// TIA Portal V17 export
// export: Created 2024-09-02T12:49:54.0325242Z, ExportSetting WithDefaults, DisplayName Totally Integrated Automation Portal, DisplayVersion V17, DisplayName TIA Portal Openness, DisplayVersion V17, DisplayName TIA Portal Version Control Interface, DisplayVersion V17, DisplayName STEP 7 Professional, DisplayVersion V17, DisplayName STEP 7 Safety, DisplayVersion V17, DisplayName WinCC Professional, DisplayVersion V17
FUNCTION_BLOCK "AnwFB_Safety"   // FB7001, F_LAD
TITLE = Safety program / Safety-Programm
{ S7_Optimized_Access := 'TRUE' }
AUTHOR : OlegFuehrus
FAMILY : SAFETY
NAME : SAFETY
VERSION : 0.1
// stored: AutoNumber false, IsIECCheckEnabled false, UDAEnableTagReadback false
   VAR
      statTrue : Bool := true;   // TRUE
      statFalse : Bool := false;   // FALSE
      HM_1_ack : Bool;   // Hilfvar Quittieren / Hilfvar Acknowledge
      HM_SK_ack_1 : Bool;   // Hilfvar Quittieren Schutzkreise / Hilfvar Acknowledge Protective circuits
      HM_FGroup_ack : Bool;   // Hilfvar Quittieren F-Baugruppen / Hilfvar Acknowledge F assemblies
      HM_LC_ack_1 : Bool;   // Hilfvar Quittieren Lichtgitter / Hilfvar Acknowledge Light grid
      Error_FDback_all { ExternalWritable := 'False'} : Bool;   // Fehler FDBack / Error FDBack
      ACK_Global { S7_SetPoint := 'True'} : ACK_GL;   // ACK Global
      EStop_1 { S7_SetPoint := 'True'} : ESTOP1;   // Not-Halt / emergency stop
      EStop_2 { S7_SetPoint := 'True'} : ESTOP1;   // Not-Halt / emergency stop
      EStop_3 { S7_SetPoint := 'True'} : ESTOP1;   // Not-Halt / emergency stop
      EStop_4 { S7_SetPoint := 'True'} : ESTOP1;   // Not-Halt / emergency stop
      EStop_5 { S7_SetPoint := 'True'} : ESTOP1;   // Not-Halt / emergency stop
      EStop_6 { S7_SetPoint := 'True'} : ESTOP1;   // Not-Halt / emergency stop
      EStop_7 { S7_SetPoint := 'True'} : ESTOP1;   // Not-Halt / emergency stop
      EStop_8 { S7_SetPoint := 'True'} : ESTOP1;   // Not-Halt / emergency stop
      LC_1 { S7_SetPoint := 'True'} : ESTOP1;   // Lichtgitter / light curtain
      LC_2 { S7_SetPoint := 'True'} : ESTOP1;   // Lichtgitter / light curtain
      LC_3 { S7_SetPoint := 'True'} : ESTOP1;   // Lichtgitter / light curtain
      LC_4 { S7_SetPoint := 'True'} : ESTOP1;   // Lichtgitter / light curtain
      LC_5 { S7_SetPoint := 'True'} : ESTOP1;   // Lichtgitter / light curtain
      LC_MUT_1 { S7_SetPoint := 'True'} : MUT_P;   // Lichtgitter mit Muting / Light curtain with muting
      LC_MUT_2 { S7_SetPoint := 'True'} : MUT_P;   // Lichtgitter mit Muting / Light curtain with muting
      LC_MUT_3 { S7_SetPoint := 'True'} : MUT_P;   // Lichtgitter mit Muting / Light curtain with muting
      LC_MUT_4 { S7_SetPoint := 'True'} : MUT_P;   // Lichtgitter mit Muting / Light curtain with muting
      LC_MUT_5 { S7_SetPoint := 'True'} : MUT_P;   // Lichtgitter mit Muting / Light curtain with muting
      SD_1 { S7_SetPoint := 'True'} : ESTOP1;   // Schutzgitter / Safety guard
      SD_2 { S7_SetPoint := 'True'} : ESTOP1;   // Schutzgitter / Safety guard
      SD_3 { S7_SetPoint := 'True'} : ESTOP1;   // Schutzgitter / Safety guard
      SD_4 { S7_SetPoint := 'True'} : ESTOP1;   // Schutzgitter / Safety guard
      SD_5 { S7_SetPoint := 'True'} : ESTOP1;   // Schutzgitter / Safety guard
      BR_1 { S7_SetPoint := 'True'} : EV1oo2DI;   // Überbrückung / Bridging
      BR_2 { S7_SetPoint := 'True'} : EV1oo2DI;   // Überbrückung / Bridging
      BR_3 { S7_SetPoint := 'True'} : EV1oo2DI;   // Überbrückung / Bridging
      BR_4 { S7_SetPoint := 'True'} : EV1oo2DI;   // Überbrückung / Bridging
      BR_5 { S7_SetPoint := 'True'} : EV1oo2DI;   // Überbrückung / Bridging
      EnblCircuit_01 { S7_SetPoint := 'True'} : FDBACK;   // Freigabekreis / Relase circuit
      EnblCircuit_02 { S7_SetPoint := 'True'} : FDBACK;   // Freigabekreis / Relase circuit
      EnblCircuit_03 { S7_SetPoint := 'True'} : FDBACK;   // Freigabekreis / Relase circuit
      EnblCircuit_04 { S7_SetPoint := 'True'} : FDBACK;   // Freigabekreis / Relase circuit
      EnblCircuit_05 { S7_SetPoint := 'True'} : FDBACK;   // Freigabekreis / Relase circuit
      EnblCircuit_06 { S7_SetPoint := 'True'} : FDBACK;   // Freigabekreis / Relase circuit
      EnblCircuit_07 { S7_SetPoint := 'True'} : FDBACK;   // Freigabekreis / Relase circuit
      EnblCircuit_08 { S7_SetPoint := 'True'} : FDBACK;   // Freigabekreis / Relase circuit
      EnblCircuit_09 { S7_SetPoint := 'True'} : FDBACK;   // Freigabekreis / Relase circuit
      EnblCircuit_10 { S7_SetPoint := 'True'} : FDBACK;   // Freigabekreis / Relase circuit
      EnblCircuit_11 { S7_SetPoint := 'True'} : FDBACK;   // Freigabekreis / Relase circuit
      EnblCircuit_12 { S7_SetPoint := 'True'} : FDBACK;   // Freigabekreis / Relase circuit
      EnblCircuit_13 { S7_SetPoint := 'True'} : FDBACK;   // Freigabekreis / Relase circuit
      EnblCircuit_14 { S7_SetPoint := 'True'} : FDBACK;   // Freigabekreis / Relase circuit
      EnblCircuit_15 { S7_SetPoint := 'True'} : FDBACK;   // Freigabekreis / Relase circuit
      SafetyZone_1 { S7_SetPoint := 'True'} : EV1oo2DI;   // Schutzbereich / Scope of protection
      SafetyZone_2 { S7_SetPoint := 'True'} : EV1oo2DI;   // Schutzbereich / Scope of protection
      SafetyZone_3 { S7_SetPoint := 'True'} : EV1oo2DI;   // Schutzbereich / Scope of protection
      SafetyZone_4 { S7_SetPoint := 'True'} : EV1oo2DI;   // Schutzbereich / Scope of protection
      SafetyZone_5 { S7_SetPoint := 'True'} : EV1oo2DI;   // Schutzbereich / Scope of protection
      EnblCircuit_delay_01 { S7_SetPoint := 'True'} : TOF;   // Freigabekreis verzoegert / Release circuit delayed
      EnblCircuit_delay_02 { S7_SetPoint := 'True'} : TOF;   // Freigabekreis verzoegert / Release circuit delayed
      EnblCircuit_delay_03 { S7_SetPoint := 'True'} : TOF;   // Freigabekreis verzoegert / Release circuit delayed
      EnblCircuit_delay_04 { S7_SetPoint := 'True'} : TOF;   // Freigabekreis verzoegert / Release circuit delayed
      EnblCircuit_delay_05 { S7_SetPoint := 'True'} : TOF;   // Freigabekreis verzoegert / Release circuit delayed
      EnblCircuit_delay_06 { S7_SetPoint := 'True'} : TOF;   // Freigabekreis verzoegert / Release circuit delayed
      EnblCircuit_delay_07 { S7_SetPoint := 'True'} : TOF;   // Freigabekreis verzoegert / Release circuit delayed
      EnblCircuit_delay_08 { S7_SetPoint := 'True'} : TOF;   // Freigabekreis verzoegert / Release circuit delayed
      EnblCircuit_delay_09 { S7_SetPoint := 'True'} : TOF;   // Freigabekreis verzoegert / Release circuit delayed
      EnblCircuit_delay_10 { S7_SetPoint := 'True'} : TOF;   // Freigabekreis verzoegert / Release circuit delayed
      EnblCircuit_delay_11 { S7_SetPoint := 'True'} : TOF;   // Freigabekreis verzoegert / Release circuit delayed
      EnblCircuit_delay_12 { S7_SetPoint := 'True'} : TOF;   // Freigabekreis verzoegert / Release circuit delayed
      EnblCircuit_delay_13 { S7_SetPoint := 'True'} : TOF;   // Freigabekreis verzoegert / Release circuit delayed
      EnblCircuit_delay_14 { S7_SetPoint := 'True'} : TOF;   // Freigabekreis verzoegert / Release circuit delayed
      EnblCircuit_delay_15 { S7_SetPoint := 'True'} : TOF;   // Freigabekreis verzoegert / Release circuit delayed
   END_VAR
   VAR_TEMP
      t_VKE0 : Bool;   // VKE0
      t_VKE1 : Bool;   // VKE1
      t_dummy : Bool;   // Dummy
      t_startcond_1 : Bool;   // Startvorrausetzung / starting prerequisite
      t_startcond_2 : Bool;
      t_fp_ack : Bool;   // Flanke Quit / Flank Quit
      t_fp_SQ_ack_2 : Bool;   // Flanke Quit Schutzkreis / Flank Quit protection circuit
      t_fp_SQ_ack_1 : Bool;   // Flanke Quit Schutzkreis / Flank Quit protection circuit
      t_fp_SQ_error_ack_2 : Bool;   // Flanke Quit Schutzkreis ohne Fehler / Flank Quit Protective circuit without fault
      t_fp_SQ_error_ack_1 : Bool;   // Flanke Quit Schutzkreis ohne Fehler / Flank Quit Protective circuit without fault
      t_fp_FGroup_ack_2 : Bool;   // Flanke Quit F-Baugruppen / Flank Quit F assemblies
      t_fp_FGroup_ack_1 : Bool;   // Flanke Quit F-Baugruppen / Flank Quit F assemblies
      t_fp_LC_ack_1 : Bool;   // Flanke Quit Lichtgitter / Flank Quit light grid
      t_EStopModule : Bool;
   END_VAR
   VAR_TEMP   // added for the SCL form of the ladder/FBD networks
      _w1 : Bool;
   END_VAR
BEGIN

REGION Network 1: VKE 0/1
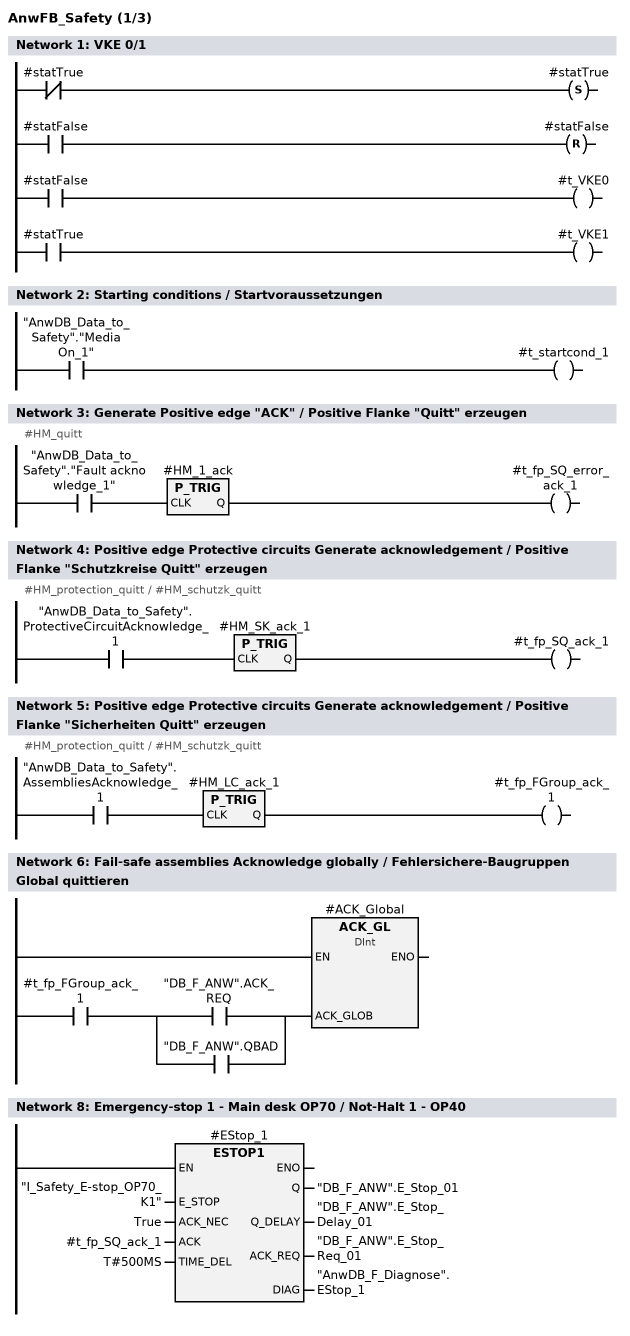
   RUNG wire#powerrail
      I_Contact( #statTrue )
      S_Coil( #statTrue )
   END_RUNG
   RUNG wire#powerrail
      Contact( #statFalse )
      R_Coil( #statFalse )
   END_RUNG
   RUNG wire#powerrail
      Contact( #statFalse )
      Coil( #t_VKE0 )
   END_RUNG
   RUNG wire#powerrail
      Contact( #statTrue )
      Coil( #t_VKE1 )
   END_RUNG
   // the same network as SCL:
   IF NOT #statTrue THEN #statTrue := TRUE; END_IF;
   IF #statFalse THEN #statFalse := FALSE; END_IF;
   #t_VKE0 := #statFalse;
   #t_VKE1 := #statTrue;
END_REGION

REGION Network 2: Starting conditions / Startvoraussetzungen
   RUNG wire#powerrail
      Contact( "AnwDB_Data_to_Safety"."Media On_1" )
      Coil( #t_startcond_1 )
   END_RUNG
   // the same network as SCL:
   #t_startcond_1 := "AnwDB_Data_to_Safety"."Media On_1";
END_REGION

REGION Network 3: Generate Positive edge "ACK" / Positive Flanke "Quitt" erzeugen
   // #HM_quitt
   RUNG wire#powerrail
      Contact( "AnwDB_Data_to_Safety"."Fault acknowledge_1" )
      P_Trig( #HM_1_ack )
      Coil( #t_fp_SQ_error_ack_1 )
   END_RUNG
   // the same network as SCL:
   #_w1 := "AnwDB_Data_to_Safety"."Fault acknowledge_1" AND NOT #HM_1_ack;   // rising edge
   #HM_1_ack := "AnwDB_Data_to_Safety"."Fault acknowledge_1";
   #t_fp_SQ_error_ack_1 := #_w1;
END_REGION

REGION Network 4: Positive edge Protective circuits Generate acknowledgement / Positive Flanke "Schutzkreise Quitt" erzeugen
   // #HM_protection_quitt / #HM_schutzk_quitt
   RUNG wire#powerrail
      Contact( "AnwDB_Data_to_Safety".ProtectiveCircuitAcknowledge_1 )
      P_Trig( #HM_SK_ack_1 )
      Coil( #t_fp_SQ_ack_1 )
   END_RUNG
   // the same network as SCL:
   #_w1 := "AnwDB_Data_to_Safety".ProtectiveCircuitAcknowledge_1 AND NOT #HM_SK_ack_1;   // rising edge
   #HM_SK_ack_1 := "AnwDB_Data_to_Safety".ProtectiveCircuitAcknowledge_1;
   #t_fp_SQ_ack_1 := #_w1;
END_REGION

REGION Network 5: Positive edge Protective circuits Generate acknowledgement / Positive Flanke "Sicherheiten Quitt" erzeugen
   // #HM_protection_quitt / #HM_schutzk_quitt
   RUNG wire#powerrail
      Contact( "AnwDB_Data_to_Safety".AssembliesAcknowledge_1 )
      P_Trig( #HM_LC_ack_1 )
      Coil( #t_fp_FGroup_ack_1 )
   END_RUNG
   // the same network as SCL:
   #_w1 := "AnwDB_Data_to_Safety".AssembliesAcknowledge_1 AND NOT #HM_LC_ack_1;   // rising edge
   #HM_LC_ack_1 := "AnwDB_Data_to_Safety".AssembliesAcknowledge_1;
   #t_fp_FGroup_ack_1 := #_w1;
END_REGION

REGION Network 6: Fail-safe assemblies Acknowledge globally / Fehlersichere-Baugruppen Global quittieren
   RUNG wire#powerrail
      { S7_Templates := "codedbool_type := DInt" } #ACK_Global.ACK_GL(ACK_GLOB := wire#w2)
   END_RUNG
   RUNG wire#powerrail
      Contact( #t_fp_FGroup_ack_1 )
      wire#w1
      Contact( "DB_F_ANW".ACK_REQ )
   END_RUNG wire#w2
   RUNG wire#w1
      Contact( "DB_F_ANW".QBAD )
   END_RUNG wire#w2
   // the same network as SCL:
   #ACK_Global(ACK_GLOB := #t_fp_FGroup_ack_1 AND ("DB_F_ANW".ACK_REQ OR "DB_F_ANW".QBAD));   // ACK_GL
END_REGION

REGION Network 7: ############# ACTUATORS ############## / ######################### AKTOREN ########################
END_REGION

REGION Network 8: Emergency-stop 1 - Main desk OP70 / Not-Halt 1 - OP40
   RUNG wire#powerrail
      #EStop_1.ESTOP1(E_STOP := "I_Safety_E-stop_OP70_K1", ACK_NEC := True, ACK := #t_fp_SQ_ack_1, TIME_DEL := T#500MS, Q => "DB_F_ANW".E_Stop_01, Q_DELAY => "DB_F_ANW".E_Stop_Delay_01, ACK_REQ => "DB_F_ANW".E_Stop_Req_01, DIAG => "AnwDB_F_Diagnose".EStop_1)
   END_RUNG
   // the same network as SCL:
   #EStop_1(E_STOP := "I_Safety_E-stop_OP70_K1",   // ESTOP1
            ACK_NEC := True,
            ACK := #t_fp_SQ_ack_1,
            TIME_DEL := T#500MS,
            Q => "DB_F_ANW".E_Stop_01,
            Q_DELAY => "DB_F_ANW".E_Stop_Delay_01,
            ACK_REQ => "DB_F_ANW".E_Stop_Req_01,
            DIAG => "AnwDB_F_Diagnose".EStop_1);
END_REGION

REGION Network 9: Emergency stop OK. / Not-Halt i.O.
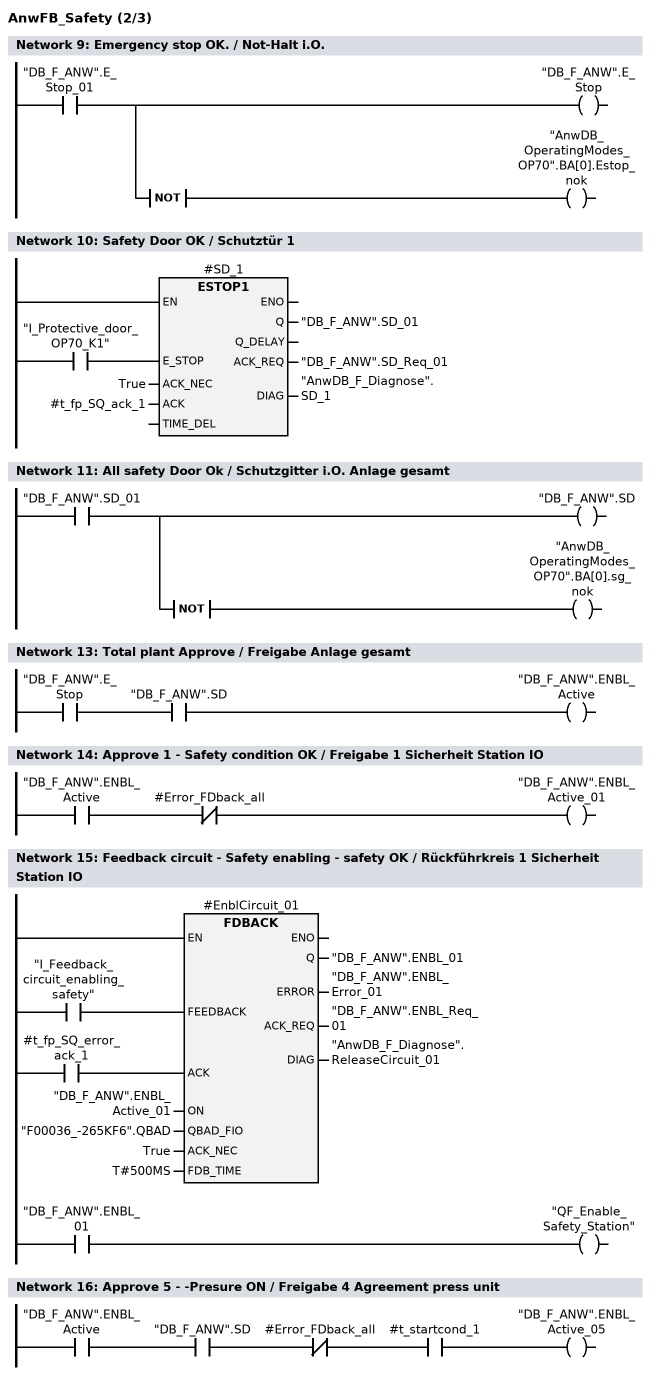
   RUNG wire#powerrail
      Contact( "DB_F_ANW".E_Stop_01 )
      wire#w1
      Coil( "DB_F_ANW".E_Stop )
   END_RUNG
   RUNG wire#w1
      Not()
      Coil( "AnwDB_OperatingModes_OP70".BA[0].Estop_nok )
   END_RUNG
   // the same network as SCL:
   "DB_F_ANW".E_Stop := "DB_F_ANW".E_Stop_01;
   "AnwDB_OperatingModes_OP70".BA[0].Estop_nok := NOT "DB_F_ANW".E_Stop_01;
END_REGION

REGION Network 10: Safety Door OK / Schutztür 1
   RUNG wire#powerrail
      #SD_1.ESTOP1(E_STOP := wire#w1, ACK_NEC := True, ACK := #t_fp_SQ_ack_1, TIME_DEL :=, Q => "DB_F_ANW".SD_01, Q_DELAY =>, ACK_REQ => "DB_F_ANW".SD_Req_01, DIAG => "AnwDB_F_Diagnose".SD_1)
   END_RUNG
   RUNG wire#powerrail
      Contact( "I_Protective_door_OP70_K1" )
   END_RUNG wire#w1
   // the same network as SCL:
   #SD_1(E_STOP := "I_Protective_door_OP70_K1",   // ESTOP1
         ACK_NEC := True,
         ACK := #t_fp_SQ_ack_1,
         Q => "DB_F_ANW".SD_01,
         ACK_REQ => "DB_F_ANW".SD_Req_01,
         DIAG => "AnwDB_F_Diagnose".SD_1);
END_REGION

REGION Network 11: All safety Door Ok / Schutzgitter i.O. Anlage gesamt
   RUNG wire#powerrail
      Contact( "DB_F_ANW".SD_01 )
      wire#w1
      Coil( "DB_F_ANW".SD )
   END_RUNG
   RUNG wire#w1
      Not()
      Coil( "AnwDB_OperatingModes_OP70".BA[0].sg_nok )
   END_RUNG
   // the same network as SCL:
   "DB_F_ANW".SD := "DB_F_ANW".SD_01;
   "AnwDB_OperatingModes_OP70".BA[0].sg_nok := NOT "DB_F_ANW".SD_01;
END_REGION

REGION Network 12: ############# PERMISIIONS ############## / ######################### FREIGABEN ########################
END_REGION

REGION Network 13: Total plant Approve / Freigabe Anlage gesamt
   RUNG wire#powerrail
      Contact( "DB_F_ANW".E_Stop )
      Contact( "DB_F_ANW".SD )
      Coil( "DB_F_ANW".ENBL_Active )
   END_RUNG
   // the same network as SCL:
   "DB_F_ANW".ENBL_Active := "DB_F_ANW".E_Stop AND "DB_F_ANW".SD;
END_REGION

REGION Network 14: Approve 1 - Safety condition OK / Freigabe 1 Sicherheit Station IO
   RUNG wire#powerrail
      Contact( "DB_F_ANW".ENBL_Active )
      I_Contact( #Error_FDback_all )
      Coil( "DB_F_ANW".ENBL_Active_01 )
   END_RUNG
   // the same network as SCL:
   "DB_F_ANW".ENBL_Active_01 := "DB_F_ANW".ENBL_Active AND NOT #Error_FDback_all;
END_REGION

REGION Network 15: Feedback circuit - Safety enabling - safety OK / Rückführkreis 1 Sicherheit Station IO
   RUNG wire#powerrail
      #EnblCircuit_01.FDBACK(FEEDBACK := wire#w1, ACK := wire#w2, ON := "DB_F_ANW".ENBL_Active_01, QBAD_FIO := "F00036_-265KF6".QBAD, ACK_NEC := True, FDB_TIME := T#500MS, Q => "DB_F_ANW".ENBL_01, ERROR => "DB_F_ANW".ENBL_Error_01, ACK_REQ => "DB_F_ANW".ENBL_Req_01, DIAG => "AnwDB_F_Diagnose".ReleaseCircuit_01)
   END_RUNG
   RUNG wire#powerrail
      Contact( "I_Feedback_circuit_enabling_safety" )
   END_RUNG wire#w1
   RUNG wire#powerrail
      Contact( #t_fp_SQ_error_ack_1 )
   END_RUNG wire#w2
   RUNG wire#powerrail
      Contact( "DB_F_ANW".ENBL_01 )
      Coil( "QF_Enable_Safety_Station" )
   END_RUNG
   // the same network as SCL:
   #EnblCircuit_01(FEEDBACK := "I_Feedback_circuit_enabling_safety",   // FDBACK
                   ACK := #t_fp_SQ_error_ack_1,
                   ON := "DB_F_ANW".ENBL_Active_01,
                   QBAD_FIO := "F00036_-265KF6".QBAD,
                   ACK_NEC := True,
                   FDB_TIME := T#500MS,
                   Q => "DB_F_ANW".ENBL_01,
                   ERROR => "DB_F_ANW".ENBL_Error_01,
                   ACK_REQ => "DB_F_ANW".ENBL_Req_01,
                   DIAG => "AnwDB_F_Diagnose".ReleaseCircuit_01);
   "QF_Enable_Safety_Station" := "DB_F_ANW".ENBL_01;
END_REGION

REGION Network 16: Approve 5 - -Presure ON / Freigabe 4 Agreement press unit
   RUNG wire#powerrail
      Contact( "DB_F_ANW".ENBL_Active )
      Contact( "DB_F_ANW".SD )
      I_Contact( #Error_FDback_all )
      Contact( #t_startcond_1 )
      Coil( "DB_F_ANW".ENBL_Active_05 )
   END_RUNG
   // the same network as SCL:
   "DB_F_ANW".ENBL_Active_05 := "DB_F_ANW".ENBL_Active AND "DB_F_ANW".SD AND NOT #Error_FDback_all AND #t_startcond_1;
END_REGION

REGION Network 17: Feedback circuit - Presure ON / Rückführkreis 2 Not Halt IO
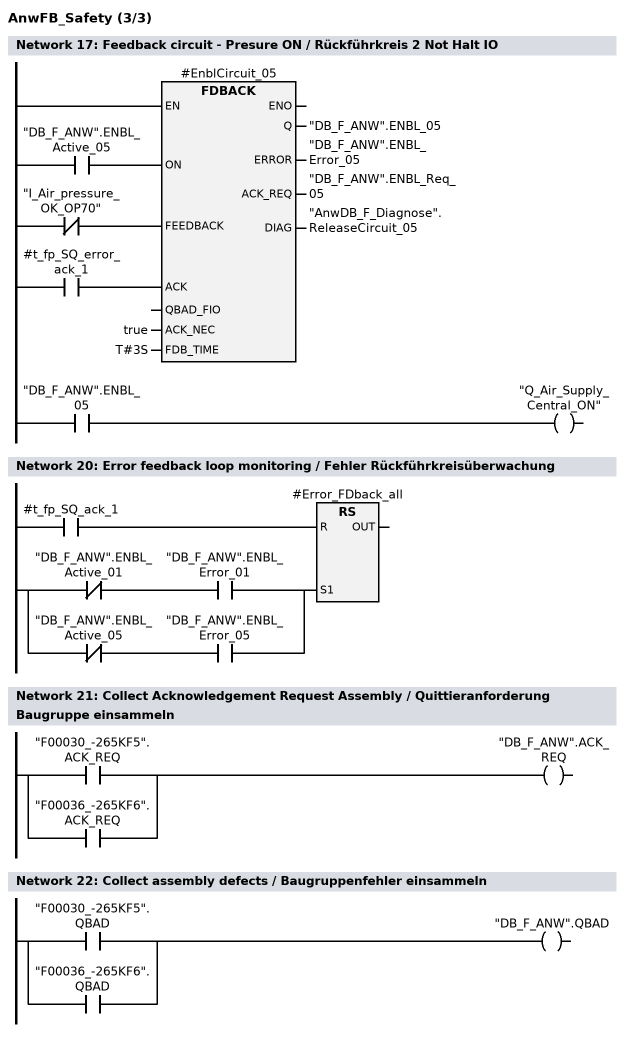
   RUNG wire#powerrail
      #EnblCircuit_05.FDBACK(ON := wire#w1, FEEDBACK := wire#w2, ACK := wire#w3, QBAD_FIO :=, ACK_NEC := true, FDB_TIME := T#3S, Q => "DB_F_ANW".ENBL_05, ERROR => "DB_F_ANW".ENBL_Error_05, ACK_REQ => "DB_F_ANW".ENBL_Req_05, DIAG => "AnwDB_F_Diagnose".ReleaseCircuit_05)
   END_RUNG
   RUNG wire#powerrail
      Contact( "DB_F_ANW".ENBL_Active_05 )
   END_RUNG wire#w1
   RUNG wire#powerrail
      I_Contact( "I_Air_pressure_OK_OP70" )
   END_RUNG wire#w2
   RUNG wire#powerrail
      Contact( #t_fp_SQ_error_ack_1 )
   END_RUNG wire#w3
   RUNG wire#powerrail
      Contact( "DB_F_ANW".ENBL_05 )
      Coil( "Q_Air_Supply_Central_ON" )
   END_RUNG
   // the same network as SCL:
   #EnblCircuit_05(ON := "DB_F_ANW".ENBL_Active_05,   // FDBACK
                   FEEDBACK := NOT "I_Air_pressure_OK_OP70",
                   ACK := #t_fp_SQ_error_ack_1,
                   ACK_NEC := true,
                   FDB_TIME := T#3S,
                   Q => "DB_F_ANW".ENBL_05,
                   ERROR => "DB_F_ANW".ENBL_Error_05,
                   ACK_REQ => "DB_F_ANW".ENBL_Req_05,
                   DIAG => "AnwDB_F_Diagnose".ReleaseCircuit_05);
   "Q_Air_Supply_Central_ON" := "DB_F_ANW".ENBL_05;
END_REGION

REGION Network 18: ############# SINAMICS ############## / ########################## SINAMICS ##############################
END_REGION

REGION Network 19: ######## USER ######### / ############# ANWENDER ##############
END_REGION

REGION Network 20: Error feedback loop monitoring / Fehler Rückführkreisüberwachung
   RUNG wire#powerrail
      Contact( #t_fp_SQ_ack_1 )
      S_RS(operand := #Error_FDback_all, s1 := wire#w1)
   END_RUNG
   RUNG wire#powerrail
      I_Contact( "DB_F_ANW".ENBL_Active_01 )
      Contact( "DB_F_ANW".ENBL_Error_01 )
   END_RUNG wire#w1
   RUNG wire#powerrail
      I_Contact( "DB_F_ANW".ENBL_Active_05 )
      Contact( "DB_F_ANW".ENBL_Error_05 )
   END_RUNG wire#w1
   // the same network as SCL:
   IF #t_fp_SQ_ack_1 THEN
       #Error_FDback_all := FALSE;   // RS flip-flop
   END_IF;
   IF (NOT "DB_F_ANW".ENBL_Active_01 AND "DB_F_ANW".ENBL_Error_01) OR (NOT "DB_F_ANW".ENBL_Active_05 AND "DB_F_ANW".ENBL_Error_05) THEN
       #Error_FDback_all := TRUE;
   END_IF;
END_REGION

REGION Network 21: Collect Acknowledgement Request Assembly / Quittieranforderung Baugruppe einsammeln
   RUNG wire#powerrail
      Contact( "F00030_-265KF5".ACK_REQ )
      wire#w1
      Coil( "DB_F_ANW".ACK_REQ )
   END_RUNG
   RUNG wire#powerrail
      Contact( "F00036_-265KF6".ACK_REQ )
   END_RUNG wire#w1
   // the same network as SCL:
   "DB_F_ANW".ACK_REQ := "F00030_-265KF5".ACK_REQ OR "F00036_-265KF6".ACK_REQ;
END_REGION

REGION Network 22: Collect assembly defects / Baugruppenfehler einsammeln
   RUNG wire#powerrail
      Contact( "F00030_-265KF5".QBAD )
      wire#w1
      Coil( "DB_F_ANW".QBAD )
   END_RUNG
   RUNG wire#powerrail
      Contact( "F00036_-265KF6".QBAD )
   END_RUNG wire#w1
   // the same network as SCL:
   "DB_F_ANW".QBAD := "F00030_-265KF5".QBAD OR "F00036_-265KF6".QBAD;
END_REGION
END_FUNCTION_BLOCK
